GLOBALCONSTANTS CommunicationPartners (* Global constants *)
  (* Standard: 61499-1 *)
  (* Version 1.0, 2025-09-06, Franz Höpfinger *)
  PACKAGE isobus::pgn;
  IMPORT isobus::pgn::ADDRESS::GLOBAL_A;
  VAR_GLOBAL CONSTANT
    GLOBAL : isobus::pgn::CF_INFO_T := (s16Handle := GLOBAL_A);
  END_VAR
END_GLOBALCONSTANTS
